{attribute 'enable_dynamic_creation'}
FUNCTION_BLOCK Circle IMPLEMENTS ITF_Shape
VAR_INPUT
	radius: INT;
END_VAR
VAR_OUTPUT
END_VAR
VAR
END_VAR


METHOD  Clone : ITF_Shape
VAR_INPUT
END_VAR
VAR_STAT
 pClone : POINTER TO Circle;	
END_VAR
pClone := __NEW(Circle);
pClone^.radius := radius;
Clone := pClone^;
__DELETE(pClone);
END_METHOD


METHOD Draw

VAR
	str : STRING;
END_VAR
str := TO_STRING(radius);

ADSLOGSTR(msgCtrlMask :=ADSLOG_MSGTYPE_HINT, msgFmtStr :='Draw circle with radius: %s', strArg := str);
END_METHOD

END_FUNCTION_BLOCK

(* stored: Version 1.1.0.1, ProductVersion 3.1.4024.12
   POU Circle: Id {7bf41376-fe79-4fc9-9b0f-cc0bfa7817da}, SpecialFunc None
   Method Clone: Id {40bc29e0-bf78-4d5d-8f5d-1f786394c013}
   Method Draw: Id {919be77b-1433-43bb-9e6d-ebea1c177f82} *)
